FUNCTION_BLOCK EQ_NeedleAxis (* Needle lift, DC motor through an L298N (IN3 up, IN4 down, ENB speed), end switches top and bottom; equipment IO: owns its IO points; commands Stop=0, Up=1, Down=2, BrakeUp=3, BrakeDown=4, Attach=5 *)
  (* Standard: 61499-2 *)
  (* Version 0.1, 2026-09-28, Project contributors, AAU Smart Production Lab *)
  PACKAGE filling;
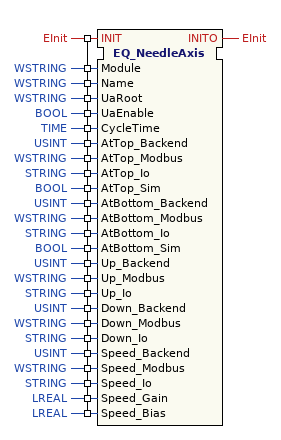
  EVENT_INPUT
    INIT : EInit WITH Module, Name, UaRoot, UaEnable, CycleTime, AtTop_Backend, AtTop_Modbus, AtTop_Io, AtTop_Sim, AtBottom_Backend, AtBottom_Modbus, AtBottom_Io, AtBottom_Sim, Up_Backend, Up_Modbus, Up_Io, Down_Backend, Down_Modbus, Down_Io, Speed_Backend, Speed_Modbus, Speed_Io, Speed_Gain, Speed_Bias;
  END_EVENT
  EVENT_OUTPUT
    INITO : EInit;
  END_EVENT
  VAR_INPUT
    Module : WSTRING;
    Name : WSTRING := "NeedleAxis";
    UaRoot : WSTRING;
    UaEnable : BOOL;
    CycleTime : TIME := T#50ms;
    AtTop_Backend : USINT := 2;
    AtTop_Modbus : WSTRING;
    AtTop_Io : STRING;
    AtTop_Sim : BOOL := FALSE;
    AtBottom_Backend : USINT := 2;
    AtBottom_Modbus : WSTRING;
    AtBottom_Io : STRING;
    AtBottom_Sim : BOOL := FALSE;
    Up_Backend : USINT := 2;
    Up_Modbus : WSTRING;
    Up_Io : STRING;
    Down_Backend : USINT := 2;
    Down_Modbus : WSTRING;
    Down_Io : STRING;
    Speed_Backend : USINT := 2;
    Speed_Modbus : WSTRING;
    Speed_Io : STRING;
    Speed_Gain : LREAL := 257.0;
    Speed_Bias : LREAL := 0.0;
  END_VAR
  FBS
    Logic : filling::EL_NeedleAxis;
    Mode : modlib::MOD_StateView;
    SubCmd : iec61499::net::SUBSCRIBE_4(QI := TRUE);
    PubState : iec61499::net::PUBLISH_3(QI := TRUE);
    PubUa : iec61499::net::PUBLISH_2;
    In_AtTop : modlib::IO_DI;
    In_AtBottom : modlib::IO_DI;
    Out_Up : modlib::IO_DO;
    Out_Down : modlib::IO_DO;
    Out_Speed : modlib::IO_AO;
    Cycle : iec61499::events::E_CYCLE;
    PhaseT : iec61499::events::E_DELAY;
  END_FBS
  EVENT_CONNECTIONS
    INIT TO Logic.INIT;
    Logic.INITO TO Mode.INIT;
    Mode.INITO TO SubCmd.INIT;
    SubCmd.INITO TO PubState.INIT;
    PubState.INITO TO PubUa.INIT;
    PubUa.INITO TO In_AtTop.INIT;
    In_AtTop.INITO TO In_AtBottom.INIT;
    In_AtBottom.INITO TO Out_Up.INIT;
    Out_Up.INITO TO Out_Down.INIT;
    Out_Down.INITO TO Out_Speed.INIT;
    Out_Speed.INITO TO Cycle.START;
    Out_Speed.INITO TO INITO;
    SubCmd.IND TO Logic.CMD;
    Mode.CHG TO Logic.MOD_CHG;
    Cycle.EO TO Logic.REFRESH;
    Cycle.EO TO In_AtTop.REQ;
    In_AtTop.CNF TO In_AtBottom.REQ;
    In_AtBottom.CNF TO Logic.SAMPLE;
    Logic.STATE TO PubState.REQ;
    Logic.STATE TO PubUa.REQ;
    Logic.DRIVE TO Out_Up.REQ;
    Out_Up.CNF TO Out_Down.REQ;
    Out_Down.CNF TO Out_Speed.REQ;
    Out_Speed.CNF TO Logic.DRIVEN;
    Logic.PHASE_START TO PhaseT.START;
    Logic.PHASE_STOP TO PhaseT.STOP;
    PhaseT.EO TO Logic.PHASE_T;
  END_CONNECTIONS
  DATA_CONNECTIONS
    Module TO Logic.Module;
    Name TO Logic.Name;
    UaRoot TO Logic.UaRoot;
    Module TO Mode.Module;
    Logic.IdCmd TO SubCmd.ID;
    Logic.IdState TO PubState.ID;
    Logic.IdPub TO PubUa.ID;
    UaEnable TO PubUa.QI;
    CycleTime TO Cycle.DT;
    SubCmd.RD_1 TO Logic.C_Holder;
    SubCmd.RD_2 TO Logic.C_Command;
    SubCmd.RD_3 TO Logic.C_Arg;
    SubCmd.RD_4 TO Logic.C_Release;
    Mode.State TO Logic.ModState;
    AtTop_Backend TO In_AtTop.Backend;
    AtTop_Modbus TO In_AtTop.ModbusId;
    AtTop_Io TO In_AtTop.IoName;
    AtTop_Sim TO In_AtTop.SimValue;
    In_AtTop.IN TO Logic.I_AtTop;
    Logic.AtTop TO PubState.SD_1;
    Logic.AtTop TO PubUa.SD_1;
    AtBottom_Backend TO In_AtBottom.Backend;
    AtBottom_Modbus TO In_AtBottom.ModbusId;
    AtBottom_Io TO In_AtBottom.IoName;
    AtBottom_Sim TO In_AtBottom.SimValue;
    In_AtBottom.IN TO Logic.I_AtBottom;
    Logic.AtBottom TO PubState.SD_2;
    Logic.AtBottom TO PubUa.SD_2;
    Logic.Holder TO PubState.SD_3;
    Up_Backend TO Out_Up.Backend;
    Up_Modbus TO Out_Up.ModbusId;
    Up_Io TO Out_Up.IoName;
    Logic.O_Up TO Out_Up.OUT;
    Down_Backend TO Out_Down.Backend;
    Down_Modbus TO Out_Down.ModbusId;
    Down_Io TO Out_Down.IoName;
    Logic.O_Down TO Out_Down.OUT;
    Speed_Backend TO Out_Speed.Backend;
    Speed_Modbus TO Out_Speed.ModbusId;
    Speed_Io TO Out_Speed.IoName;
    Logic.O_Speed TO Out_Speed.OUT;
    Logic.E_Speed TO Out_Speed.EN;
    Speed_Gain TO Out_Speed.Gain;
    Speed_Bias TO Out_Speed.Bias;
    Logic.PhaseDT TO PhaseT.DT;
  END_CONNECTIONS
END_FUNCTION_BLOCK
